// TwinCAT 3 PLC project StetigerTemperaturRegler
// ProgramVersion: 3.1.4022.1
// libraries:
//   Tc2_ControllerToolbox, * (Beckhoff Automation GmbH)
//   Tc2_Standard, * (Beckhoff Automation GmbH)
//   Tc2_System, * (Beckhoff Automation GmbH)
//   Tc2_TempController, * (Beckhoff Automation GmbH)
//   Tc2_Utilities, * (Beckhoff Automation GmbH)
//   Tc3_Module, * (Beckhoff Automation GmbH)
// project tree:
//   GVLs/ AN.TcGVL (not stored), DIO.TcGVL (not stored), dSub.TcGVL (not stored)
//   / PlcTask.TcTTO (not stored)
//   POUs/ MAIN.TcPOU, StetigerTemperaturRegler.TcPOU
// real-time tasks:
//   TASK PlcTask: cycle T#10ms, priority 20, ADS port 350
// motion (NC):
//   TASK NC-Task 1 SAF: cycle T#2ms, priority 4, ADS port 501
//   TASK NC-Task 1 SVB: cycle T#10ms, priority 8, ADS port 511
//   AXIS Axis 1 (id 1)
//     OtherSettings: AllowMotionCmdToSlave=true
//     encoder EncType=4
//       EncPara: MaxCount=#x0000ffff
//         Inc: RefSoftSyncMask=#x0000ffff
//     drive DrvType=24
//       Analog: ScaleFactorActTorque=0.1
//       TimeComp: TaskDelayCycles=1
//     controller CtrType=1
//       CtrPara: PriorControlFactor=1
//         Observer: BandWidth=20
//   AXIS Axis 2 (id 2)
//     OtherSettings: AllowMotionCmdToSlave=true
//     encoder EncType=4
//       EncPara: MaxCount=#x0000ffff
//         Inc: RefSoftSyncMask=#x0000ffff
//     drive DrvType=24
//       Analog: ScaleFactorActTorque=0.1
//       TimeComp: TaskDelayCycles=1
//     controller CtrType=1
//       CtrPara: PriorControlFactor=1
//         Observer: BandWidth=20
//   AXIS Axis 3 (id 3)
//     OtherSettings: AllowMotionCmdToSlave=true
//     encoder EncType=4
//       EncPara: MaxCount=#x0000ffff
//     drive DrvType=23
//       Analog: ScaleFactorActTorque=0.1
//       TimeComp: TaskDelayCycles=1
//     controller CtrType=1
//       CtrPara: PriorControlFactor=1
//         Observer: BandWidth=20
//   AXIS Axis 4 (id 4)
//     OtherSettings: AllowMotionCmdToSlave=true
//     encoder EncType=4
//       EncPara: MaxCount=#x0000ffff
//     drive DrvType=23
//       Analog: ScaleFactorActTorque=0.1
//       TimeComp: TaskDelayCycles=1
//     controller CtrType=1
//       CtrPara: PriorControlFactor=1
//         Observer: BandWidth=20
//   AXIS Axis 5 (id 5)
//     OtherSettings: AllowMotionCmdToSlave=true
//     encoder EncType=19
//       EncPara: MaxCount=#xffffffff
//     drive DrvType=16
//       DrvPara: MaxCount=#xffffffff
//         Analog: ScaleFactorActTorque=0.1
//         TimeComp: TaskDelayCycles=1
//     controller CtrType=1
//       CtrPara: PriorControlFactor=1
//         Observer: BandWidth=20
//   AXIS Axis 6 (id 6)
//     OtherSettings: AllowMotionCmdToSlave=true
//     encoder EncType=19
//       EncPara: MaxCount=#xffffffff
//     drive DrvType=16
//       DrvPara: MaxCount=#xffffffff
//         Analog: ScaleFactorActTorque=0.1
//         TimeComp: TaskDelayCycles=1
//     controller CtrType=1
//       CtrPara: PriorControlFactor=1
//         Observer: BandWidth=20
// I/O:
//   DEVICE Device 1 (EtherCAT), AmsNetId 5.35.139.20.2.1
//     Term 1 (EK1200) [EK1200-5000 EtherCAT Power supply (2A E-Bus)]
//       Term 2 (EL1809) [EL1809 16Ch. Dig. Input 24V, 3ms]
//       Term 3 (EL1809) [EL1809 16Ch. Dig. Input 24V, 3ms]
//       Term 4 (EL2809) [EL2809 16Ch. Dig. Output 24V, 0.5A]
//       Term 5 (EL2809) [EL2809 16Ch. Dig. Output 24V, 0.5A]
//       Term 6 (EL3064) [EL3064 4Ch. Ana. Input 0-10V]
//       Term 7 (EL4034) [EL4034 4Ch. Ana. Output +/-10V, 12bit]
//       Term 8 (EL7031) [EL7031 1Ch. Stepper motor output stage (24V, 1.5A)]
//       Term 9 (EL7031) [EL7031 1Ch. Stepper motor output stage (24V, 1.5A)]
//       Term 10 (EL7332) [EL7332 2Ch. DC motor output stage (24V, 1.5A)]
//       Term 11 (EL7201-0010) [EL7201-0010 1Ch. MDP742 Servo motor output stage with OCT (50V, 4A)]
//       Term 12 (EL7201-0010) [EL7201-0010 1Ch. MDP742 Servo motor output stage with OCT (50V, 4A)]
//       Term 26 (EL6090) [EL6090 Display terminal]
//       Term 27 (EK1110) [EK1110 EtherCAT extension]
// variable links:
//   NC-Task 1 SAF/Axes/Axis 1 <-> Device 1 (EtherCAT)/Term 1 (EK1200)/Term 8 (EL7031)
//     Drive/Inputs/In/nState1 @bit 3 <-> STM Status/Status/Error
//     Drive/Inputs/In/nState1 @bit 5 <-> STM Status/Status/Moving negative
//     Drive/Inputs/In/nState1 @bit 4 <-> STM Status/Status/Moving positive
//     Drive/Inputs/In/nState1 @bit 1 <-> STM Status/Status/Ready
//     Drive/Inputs/In/nState1 <-> STM Status/Status/Ready to enable
//     Drive/Inputs/In/nState1 @bit 6 <-> STM Status/Status/Torque reduced
//     Drive/Inputs/In/nState1 @bit 2 <-> STM Status/Status/Warning
//     Drive/Inputs/In/nState2 @bit 3 <-> STM Status/Status/Digital input 1
//     Drive/Inputs/In/nState2 @bit 4 <-> STM Status/Status/Digital input 2
//     Drive/Inputs/In/nState2 @bit 5 <-> STM Status/Status/Sync error
//     Drive/Inputs/In/nState2 @bit 7 <-> STM Status/Status/TxPDO Toggle
//     Drive/Inputs/In/nState4 @bit 1 <-> WcState/InputToggle
//     Drive/Inputs/In/nState4 <-> WcState/WcState
//     Drive/Outputs/Out/nCtrl1 <-> STM Control/Control/Enable
//     Drive/Outputs/Out/nCtrl1 @bit 2 <-> STM Control/Control/Reduce torque
//     Drive/Outputs/Out/nCtrl1 @bit 1 <-> STM Control/Control/Reset
//     Drive/Outputs/Out/nDataOut2[0] <-> STM Velocity/Velocity
//     Enc/Inputs/In/nDataIn1[0] <-> ENC Status compact/Counter value
//     Enc/Inputs/In/nDataIn2[0] <-> ENC Status compact/Latch value
//     Enc/Inputs/In/nState1 @bit 4 <-> ENC Status compact/Status/Counter overflow
//     Enc/Inputs/In/nState1 @bit 3 <-> ENC Status compact/Status/Counter underflow
//     Enc/Inputs/In/nState1 @bit 1 <-> ENC Status compact/Status/Latch extern valid
//     Enc/Inputs/In/nState1 @bit 2 <-> ENC Status compact/Status/Set counter done
//     Enc/Inputs/In/nState2 @bit 4 <-> ENC Status compact/Status/Status of extern latch
//     Enc/Inputs/In/nState2 @bit 5 <-> ENC Status compact/Status/Sync error
//     Enc/Inputs/In/nState2 @bit 7 <-> ENC Status compact/Status/TxPDO Toggle
//     Enc/Inputs/In/nState4 @bit 1 <-> WcState/InputToggle
//     Enc/Inputs/In/nState4 <-> WcState/WcState
//     Enc/Outputs/Out/nCtrl1 @bit 3 <-> ENC Control compact/Control/Enable latch extern on negative edge
//     Enc/Outputs/Out/nCtrl1 @bit 1 <-> ENC Control compact/Control/Enable latch extern on positive edge
//     Enc/Outputs/Out/nCtrl1 @bit 2 <-> ENC Control compact/Control/Set counter
//     Enc/Outputs/Out/nDataOut1[0] <-> ENC Control compact/Set counter value
//   NC-Task 1 SAF/Axes/Axis 2 <-> Device 1 (EtherCAT)/Term 1 (EK1200)/Term 9 (EL7031)
//     Drive/Inputs/In/nState1 @bit 3 <-> STM Status/Status/Error
//     Drive/Inputs/In/nState1 @bit 5 <-> STM Status/Status/Moving negative
//     Drive/Inputs/In/nState1 @bit 4 <-> STM Status/Status/Moving positive
//     Drive/Inputs/In/nState1 @bit 1 <-> STM Status/Status/Ready
//     Drive/Inputs/In/nState1 <-> STM Status/Status/Ready to enable
//     Drive/Inputs/In/nState1 @bit 6 <-> STM Status/Status/Torque reduced
//     Drive/Inputs/In/nState1 @bit 2 <-> STM Status/Status/Warning
//     Drive/Inputs/In/nState2 @bit 3 <-> STM Status/Status/Digital input 1
//     Drive/Inputs/In/nState2 @bit 4 <-> STM Status/Status/Digital input 2
//     Drive/Inputs/In/nState2 @bit 5 <-> STM Status/Status/Sync error
//     Drive/Inputs/In/nState2 @bit 7 <-> STM Status/Status/TxPDO Toggle
//     Drive/Inputs/In/nState4 @bit 1 <-> WcState/InputToggle
//     Drive/Inputs/In/nState4 <-> WcState/WcState
//     Drive/Outputs/Out/nCtrl1 <-> STM Control/Control/Enable
//     Drive/Outputs/Out/nCtrl1 @bit 2 <-> STM Control/Control/Reduce torque
//     Drive/Outputs/Out/nCtrl1 @bit 1 <-> STM Control/Control/Reset
//     Drive/Outputs/Out/nDataOut2[0] <-> STM Velocity/Velocity
//     Enc/Inputs/In/nDataIn1[0] <-> ENC Status compact/Counter value
//     Enc/Inputs/In/nDataIn2[0] <-> ENC Status compact/Latch value
//     Enc/Inputs/In/nState1 @bit 4 <-> ENC Status compact/Status/Counter overflow
//     Enc/Inputs/In/nState1 @bit 3 <-> ENC Status compact/Status/Counter underflow
//     Enc/Inputs/In/nState1 @bit 1 <-> ENC Status compact/Status/Latch extern valid
//     Enc/Inputs/In/nState1 @bit 2 <-> ENC Status compact/Status/Set counter done
//     Enc/Inputs/In/nState2 @bit 4 <-> ENC Status compact/Status/Status of extern latch
//     Enc/Inputs/In/nState2 @bit 5 <-> ENC Status compact/Status/Sync error
//     Enc/Inputs/In/nState2 @bit 7 <-> ENC Status compact/Status/TxPDO Toggle
//     Enc/Inputs/In/nState4 @bit 1 <-> WcState/InputToggle
//     Enc/Inputs/In/nState4 <-> WcState/WcState
//     Enc/Outputs/Out/nCtrl1 @bit 3 <-> ENC Control compact/Control/Enable latch extern on negative edge
//     Enc/Outputs/Out/nCtrl1 @bit 1 <-> ENC Control compact/Control/Enable latch extern on positive edge
//     Enc/Outputs/Out/nCtrl1 @bit 2 <-> ENC Control compact/Control/Set counter
//     Enc/Outputs/Out/nDataOut1[0] <-> ENC Control compact/Set counter value
//   NC-Task 1 SAF/Axes/Axis 3 <-> Device 1 (EtherCAT)/Term 1 (EK1200)/Term 10 (EL7332)
//     Drive/Inputs/In/nState1 @bit 3 <-> DCM Status Channel 1/Status/Error
//     Drive/Inputs/In/nState1 @bit 5 <-> DCM Status Channel 1/Status/Moving negative
//     Drive/Inputs/In/nState1 @bit 4 <-> DCM Status Channel 1/Status/Moving positive
//     Drive/Inputs/In/nState1 @bit 1 <-> DCM Status Channel 1/Status/Ready
//     Drive/Inputs/In/nState1 <-> DCM Status Channel 1/Status/Ready to enable
//     Drive/Inputs/In/nState1 @bit 6 <-> DCM Status Channel 1/Status/Torque reduced
//     Drive/Inputs/In/nState1 @bit 2 <-> DCM Status Channel 1/Status/Warning
//     Drive/Inputs/In/nState2 @bit 3 <-> DCM Status Channel 1/Status/Digital input 1
//     Drive/Inputs/In/nState2 @bit 4 <-> DCM Status Channel 1/Status/Digital input 2
//     Drive/Inputs/In/nState2 @bit 5 <-> DCM Status Channel 1/Status/Sync error
//     Drive/Inputs/In/nState2 @bit 7 <-> DCM Status Channel 1/Status/TxPDO Toggle
//     Drive/Inputs/In/nState4 @bit 1 <-> WcState/InputToggle
//     Drive/Inputs/In/nState4 <-> WcState/WcState
//     Drive/Outputs/Out/nCtrl1 <-> DCM Control Channel 1/Control/Enable
//     Drive/Outputs/Out/nCtrl1 @bit 2 <-> DCM Control Channel 1/Control/Reduce torque
//     Drive/Outputs/Out/nCtrl1 @bit 1 <-> DCM Control Channel 1/Control/Reset
//     Drive/Outputs/Out/nDataOut2[0] <-> DCM Velocity Channel 1/Velocity
//   NC-Task 1 SAF/Axes/Axis 4 <-> Device 1 (EtherCAT)/Term 1 (EK1200)/Term 10 (EL7332)
//     Drive/Inputs/In/nState1 @bit 3 <-> DCM Status Channel 2/Status/Error
//     Drive/Inputs/In/nState1 @bit 5 <-> DCM Status Channel 2/Status/Moving negative
//     Drive/Inputs/In/nState1 @bit 4 <-> DCM Status Channel 2/Status/Moving positive
//     Drive/Inputs/In/nState1 @bit 1 <-> DCM Status Channel 2/Status/Ready
//     Drive/Inputs/In/nState1 <-> DCM Status Channel 2/Status/Ready to enable
//     Drive/Inputs/In/nState1 @bit 6 <-> DCM Status Channel 2/Status/Torque reduced
//     Drive/Inputs/In/nState1 @bit 2 <-> DCM Status Channel 2/Status/Warning
//     Drive/Inputs/In/nState2 @bit 3 <-> DCM Status Channel 2/Status/Digital input 1
//     Drive/Inputs/In/nState2 @bit 4 <-> DCM Status Channel 2/Status/Digital input 2
//     Drive/Inputs/In/nState2 @bit 5 <-> DCM Status Channel 2/Status/Sync error
//     Drive/Inputs/In/nState2 @bit 7 <-> DCM Status Channel 2/Status/TxPDO Toggle
//     Drive/Inputs/In/nState4 @bit 1 <-> WcState/InputToggle
//     Drive/Inputs/In/nState4 <-> WcState/WcState
//     Drive/Outputs/Out/nCtrl1 <-> DCM Control Channel 2/Control/Enable
//     Drive/Outputs/Out/nCtrl1 @bit 2 <-> DCM Control Channel 2/Control/Reduce torque
//     Drive/Outputs/Out/nCtrl1 @bit 1 <-> DCM Control Channel 2/Control/Reset
//     Drive/Outputs/Out/nDataOut2[0] <-> DCM Velocity Channel 2/Velocity
//   NC-Task 1 SAF/Axes/Axis 5 <-> Device 1 (EtherCAT)/Term 1 (EK1200)/Term 11 (EL7201-0010)
//     Drive/Inputs/In/nDcOutputTime <-> InfoData/DcOutputShift
//     Drive/Inputs/In/nState1 <-> DRV Statusword/Statusword
//     Drive/Inputs/In/nState2 <-> DRV Statusword/Statusword @bit 8
//     Drive/Inputs/In/nState4 @bit 1 <-> WcState/InputToggle
//     Drive/Inputs/In/nState4 <-> WcState/WcState
//     Drive/Outputs/Out/nCtrl1 <-> DRV Controlword/Controlword
//     Drive/Outputs/Out/nCtrl2 <-> DRV Controlword/Controlword @bit 8
//     Drive/Outputs/Out/nDataOut2 <-> DRV Target velocity/Target velocity
//     Enc/Inputs/In/nDataIn1 <-> FB Position/Position
//     Enc/Inputs/In/nDcInputTime <-> InfoData/DcInputShift
//     Enc/Inputs/In/nState4 @bit 1 <-> WcState/InputToggle
//     Enc/Inputs/In/nState4 <-> WcState/WcState
//   NC-Task 1 SAF/Axes/Axis 6 <-> Device 1 (EtherCAT)/Term 1 (EK1200)/Term 12 (EL7201-0010)
//     Drive/Inputs/In/nDcOutputTime <-> InfoData/DcOutputShift
//     Drive/Inputs/In/nState1 <-> DRV Statusword/Statusword
//     Drive/Inputs/In/nState2 <-> DRV Statusword/Statusword @bit 8
//     Drive/Inputs/In/nState4 @bit 1 <-> WcState/InputToggle
//     Drive/Inputs/In/nState4 <-> WcState/WcState
//     Drive/Outputs/Out/nCtrl1 <-> DRV Controlword/Controlword
//     Drive/Outputs/Out/nCtrl2 <-> DRV Controlword/Controlword @bit 8
//     Drive/Outputs/Out/nDataOut2 <-> DRV Target velocity/Target velocity
//     Enc/Inputs/In/nDataIn1 <-> FB Position/Position
//     Enc/Inputs/In/nDcInputTime <-> InfoData/DcInputShift
//     Enc/Inputs/In/nState4 @bit 1 <-> WcState/InputToggle
//     Enc/Inputs/In/nState4 <-> WcState/WcState
//   StetigerTemperaturRegler/StetigerTemperaturRegler Instance <-> Device 1 (EtherCAT)/Term 1 (EK1200)/Term 2 (EL1809)
//     PlcTask Inputs/dSub.B1 <-> Channel 1/Input
//     PlcTask Inputs/dSub.B2 <-> Channel 2/Input
//     PlcTask Inputs/dSub.S1 <-> Channel 4/Input
//     PlcTask Inputs/dSub.S10 <-> Channel 12/Input
//     PlcTask Inputs/dSub.S11 <-> Channel 13/Input
//     PlcTask Inputs/dSub.S2 <-> Channel 3/Input
//     PlcTask Inputs/dSub.S3 <-> Channel 6/Input
//     PlcTask Inputs/dSub.S4 <-> Channel 5/Input
//     PlcTask Inputs/dSub.S5 <-> Channel 8/Input
//     PlcTask Inputs/dSub.S6 <-> Channel 7/Input
//     PlcTask Inputs/dSub.S7 <-> Channel 10/Input
//     PlcTask Inputs/dSub.S8 <-> Channel 9/Input
//     PlcTask Inputs/dSub.S9 <-> Channel 11/Input
//   StetigerTemperaturRegler/StetigerTemperaturRegler Instance <-> Device 1 (EtherCAT)/Term 1 (EK1200)/Term 3 (EL1809)
//     PlcTask Inputs/DIO.DI_{1..16} <-> Channel {1..16}/Input  (16 links)
//   StetigerTemperaturRegler/StetigerTemperaturRegler Instance <-> Device 1 (EtherCAT)/Term 1 (EK1200)/Term 4 (EL2809)
//     PlcTask Outputs/dSub.P{1..4} <-> Channel {3..6}/Output  (4 links)
//     PlcTask Outputs/dSub.Q1 <-> Channel 1/Output
//     PlcTask Outputs/dSub.Q2 <-> Channel 2/Output
//   StetigerTemperaturRegler/StetigerTemperaturRegler Instance <-> Device 1 (EtherCAT)/Term 1 (EK1200)/Term 5 (EL2809)
//     PlcTask Outputs/DIO.DQ_{1..16} <-> Channel {1..16}/Output  (16 links)
//   StetigerTemperaturRegler/StetigerTemperaturRegler Instance <-> Device 1 (EtherCAT)/Term 1 (EK1200)/Term 6 (EL3064)
//     PlcTask Inputs/AN.AI_1 <-> AI Standard Channel 3/Value
//     PlcTask Inputs/AN.AI_2 <-> AI Standard Channel 4/Value
//     PlcTask Inputs/dSub.AI_0 <-> AI Standard Channel 1/Value
//     PlcTask Inputs/dSub.AI_1 <-> AI Standard Channel 2/Value
//   StetigerTemperaturRegler/StetigerTemperaturRegler Instance <-> Device 1 (EtherCAT)/Term 1 (EK1200)/Term 7 (EL4034)
//     PlcTask Outputs/AN.AQ_1 <-> AO Outputs Channel 3/Analog output
//     PlcTask Outputs/AN.AQ_2 <-> AO Outputs Channel 4/Analog output
//     PlcTask Outputs/dSub.AQ_0 <-> AO Outputs Channel 1/Analog output

// ---- POUs/MAIN.TcPOU
PROGRAM MAIN
VAR

END_VAR

StetigerTemperaturRegler();

END_PROGRAM

// ---- POUs/StetigerTemperaturRegler.TcPOU
PROGRAM StetigerTemperaturRegler
VAR
	
		eCTRL_Mode 				: E_CTRL_MODE := eCTRL_MODE_Tune; 	(*   eCTRL_MODE_TUNE  ;*)
		bSelSetpoint			: BOOL	:= FALSE;
		
		fW						: LREAL;						(* setpoint *)
		fW1						: LREAL := 70;					(* first setpoint *)
		fW2						: LREAL := 35.0;				(* second setpoint - standby setpoint*)
		fY						: LREAL;						(* control value *)
		fX						: LREAL;						(* actual value from simulated process *)
		bYPWMPos				: BOOL;
		bYPWMNeg				: BOOL;
		
		bNoise					: BOOL;
		bError 					: BOOL;
		eErrorId 				: E_CTRL_ErrorCodes;
		
		stControllerParameter	: ST_CTRL_TempCtrlParameter := (		
		
		(* general parameters 													 *)
		iMode					:= 1,											(* 1=heating, 2=cooling, 3=heating&cooling *)
		iReactionOnFailure		:= eCTRL_ReactionOnFailure_StopController,		(* 0=controller off, 1=manual op, 2=yMin, 3=yMax *)
	
		bSelCtrlParameterSet	:= FALSE,										(* FALSE = internal set, TRUE = external set *)
	
		dwAlarmSupp				:= 16#0000EFFF,									(* alarm suppression *)
		tCtrlCycleTime			:= T#500MS,										(* controller cycle time *)
		tTaskCycleTime			:= T#10MS,										(* plc task cycle time *)
		
		(* tuning parameters 													 *)
		iTuningMode				:= 1,											(* only heating, only cooling, first heating then cooling or vice versa *)
	
		tTuneStabilisation		:= T#20S,										(* wait for a stable system *)
	
		fEndTunePercentHeating	:= 80.0,										(* switch to closed loop control when X > 0.8*W *)
		fYTuneHeating			:= 16000.0,										(* step change while tuning operation *)
		fYStableHeating			:= 0.0,											(* tuning operation *)
	
		fEndTunePercentCooling	:= 20.0,										(* switch to closed loop control when X < 0.2*W *)
		fYTuneCooling			:= 0.0,											(* step change while tuning operation *)
		fYStableCooling			:= 0.0,											(* tuning operation *)
		fScalingFactor			:= 1.0,											(* Scaling factor for KP heating/cooling *)
		
		(* setpoint parameters 													 *)
		fWMin					:= 0.0,											(* lower limit *)
		fWMax					:= 300.0,										(* upper limit *)
	
		(* start up *)
		bEnableSoftStart		:= FALSE,										(* FALSE = no soft start, TRUE = soft start *)
		bEnableRamping			:= FALSE,										(* FALSE = no ramping, TRUE = ramping *)
	
		fWStartUp				:= 0.0,											(* soft start plateau setpoint *)
		tStartUp				:= T#0MS,										(* soft start waiting time*)
		bStartUpRamping			:= FALSE,										(* enable ramping while start up phase *)
		fWStartUpVeloPos		:= 1.0,											(* max gradient for increasing setpoint in start up phase*)
		fWStartUpVeloNeg		:= 1.0,											(* max gradient for decreasing setpoint in start up phase *)
	
		fWVeloPos				:= 1.0,											(* max gradient for increasing setpoint *)
		fWVeloNeg				:= 1.0,											(* max gradient for decreasing setpoint *)	
	
		(* actual value parameters     											 *)
		bFilter 				:= FALSE,
		tFilter					:= T#0S,
		
		(* deadband parameters     												 *)
		bDeadband				:= FALSE,
		fEDeadband				:= 0.0,											(* deadband *)
		
		(* control value parameters     										 *)
		fYMin					:= 0.0,											(* lower limit *)
		fYMax					:= 16000.0,										(* upper limit *)
		fYManual				:= 0.0,									 		(* manual operation*)
		fYOnFailure				:= 0.0,											(* control value on failure *)
	
		tPWMCycleTime			:= t#1s,										(* PWM: period *)
		tPWMMinOffTime			:= t#0s,										(* PWM: min off time *)
		tPWMMinOnTime			:= t#0s,										(* PWM: min on time *)
		tPWMWaitingTime			:= t#0s,										(* PWM: min waiting time *) (* not yet implemented !!!!*)
	
		fYThresholdOff			:= 0.0,											(* 3-Point: Off threshold *)
		fYThresholdOn			:= 0.0,											(* 3-Point: On threshold *)
	
		nCyclesForSwitchOver	:= 100,
	
		(* controller settings			     									 *)
		bEnablePreController 	:= FALSE,										(* enable precontroller *)
		bEnableZones 			:= FALSE,										(* enable zone around setpoint with open loop control *)
		bEnableCVFilter 		:= FALSE,										(* enable filter for CV (type see iFilterType) *)
		iFilterType 			:= E_FilterType_FIRSTORDER,			 			(* filtertype of CV filter *)
		iControllerType 		:= eCTRL_ControllerType_PID,					(* used controller normally PID *)
		
		
		(* min max temperatures	     											 *)
		TempLow					:= -5.0,
		TempLowLow				:= -10.0,
		TempHigh				:= 5.0,
		TempHighHigh			:= 10.0,
		TempAbsoluteHigh		:= 300.0,
		TempAbsoluteLow			:= 0.0,	
		
		(* internal tuning parameters *)
		fTuneKp					:= 1.2,
		fTuneTn					:= 2.0,
		fTuneTv					:= 0.42,
		fTuneTd					:= 0.25
		);
	
	fbTempController			: FB_CTRL_TempController;
	
	fbCtrlParameter				: FB_CTRL_CtrlParameter;
	stController				: ST_CTRL_ParaController;
	
	(* Debug *)
	fMaxOvershoot			: LREAL;
	tStartUpTime			: TIME;
	eCtrlState				: E_CTRL_STATE;	
	
	fw_Scope : LREAL;
	fX_Scope: LREAL;
	fY_Scope: LREAL;
	fActualValue: FLOAT;
END_VAR

(* Select setpoint *)
IF bSelSetpoint THEN
	fW := fW2;
ELSE
	fW := fW1;
END_IF


fActualValue := AN.AI_1;
fActualValue := fActualValue / 326;

(* Start controller *)
fbTempController(
					eCtrlMode				:= eCTRL_Mode, 
					bSelSetpoint			:= bSelSetpoint, 
					fW1						:= fW1, 
					fW2						:= fW2, 
					fX						:= fActualValue,		// Add measured temperature here 
					fYManual				:= , 
					bOpenThermocouple		:= FALSE, 
					bReverseThermocouple	:= FALSE, 
					bBackVoltage			:= FALSE, 
					bLeakage				:= FALSE, 
					bShortCircuit			:= FALSE, 
					bOpenCircuit			:= FALSE, 
					sParaControllerExternal	:= stController, 
					sControllerParameter	:= stControllerParameter, 
					);
					 
(* Analog output *)			
fY := fbTempController.fYAnalog;

(* Digital (PWM) output *)
bYPWMPos := fbTempController.bYPWMPos;
bYPWMNeg := fbTempController.bYPWMNeg;

bError := fbTempController.bError;
eErrorId := fbTempController.eErrorId;

(* Choose set of controller parameters *)
IF fbTempController.eCtrlState = eCTRL_STATE_TUNED THEN
	eCTRL_Mode := eCTRL_MODE_ACTIVE;	
END_IF


(* Debug *)
fMaxOvershoot := fbTempController.fMaxOverShoot;
tStartUpTime := fbTempController.tStartUpTime;

(* Scope *)
fW_Scope := fW;
fX_Scope := fActualValue;
fY_Scope := fY;

(*Ausgang*)
AN.AQ_1 :=  LREAL_TO_INT(fY);	// 0 - 16.000 digit

END_PROGRAM
